% RSLogix 500 project PRJ_OUM_BAK033.RSS, saved by version 8.30.00.16 %
PROJECT "PRJ_OUM"    % processor: MicroLogix 1000 %

PROGRAM FILES
  LAD 2 "MAIN_PROG"  14 rungs
  LAD 3 "USER_FAULT"  1 rungs
  LAD 4 "HSC_INT"  1 rungs
  LAD 5 "STI_INT"  1 rungs
  LAD 6, 7, 8, 9, 10, 11, 12, 13, 14, 15, 16: only END

DATA FILES
  O0 OUTPUT  1 elements
  I1 INPUT  2 elements
  S2 STATUS  33 elements
  B3 BINARY  32 elements
  T4 TIMER  40 elements
  C5 COUNTER  32 elements
  R6 CONTROL  16 elements
  N7 INTEGER  105 elements

LADDER 2 "MAIN_PROG"
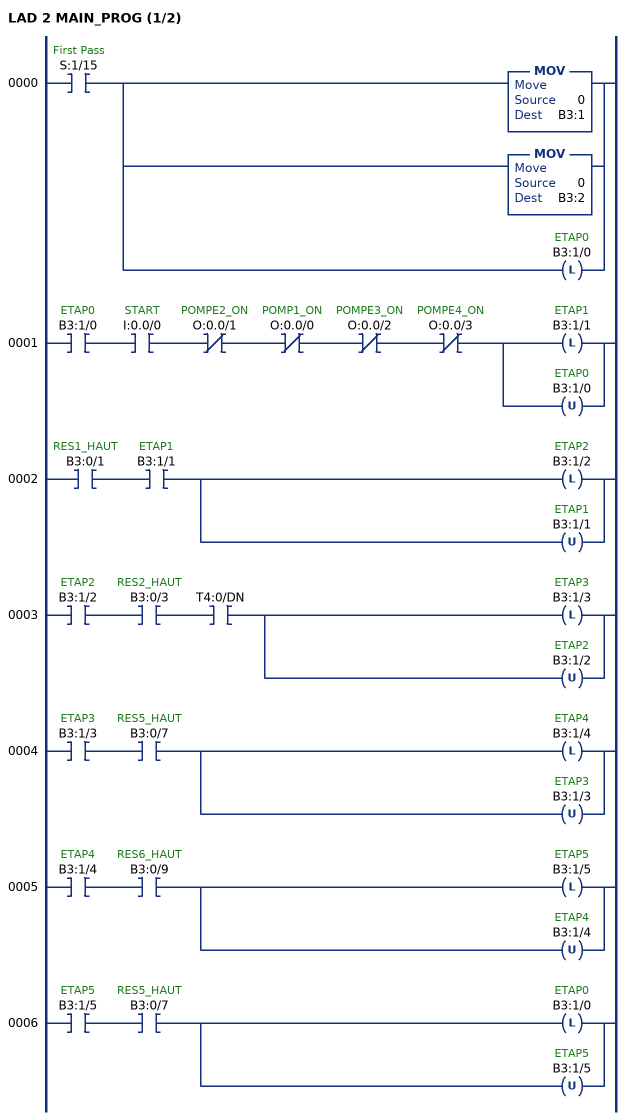
% Rung: 0 %
SOR XIC S:1/15 BST MOV 0 B3:1 NXB BST MOV 0 B3:2 NXB OTL B3:1/0 BND BND EOR
%   S:1/15  "First Pass" %
%   B3:1/0  ETAP0 %
% Rung: 1 %
SOR XIC B3:1/0 XIC I:0.0/0 XIO O:0.0/1 XIO O:0.0/0 XIO O:0.0/2 XIO O:0.0/3 BST OTL B3:1/1 NXB OTU B3:1/0 BND EOR
%   B3:1/0  ETAP0 %
%   I:0.0/0  START %
%   O:0.0/1  POMPE2_ON %
%   O:0.0/0  POMP1_ON %
%   O:0.0/2  POMPE3_ON %
%   O:0.0/3  POMPE4_ON %
%   B3:1/1  ETAP1 %
% Rung: 2 %
SOR XIC B3:0/1 XIC B3:1/1 BST OTL B3:1/2 NXB OTU B3:1/1 BND EOR
%   B3:0/1  RES1_HAUT %
%   B3:1/1  ETAP1 %
%   B3:1/2  ETAP2 %
% Rung: 3 %
SOR XIC B3:1/2 XIC B3:0/3 XIC T4:0/DN BST OTL B3:1/3 NXB OTU B3:1/2 BND EOR
%   B3:1/2  ETAP2 %
%   B3:0/3  RES2_HAUT %
%   B3:1/3  ETAP3 %
% Rung: 4 %
SOR XIC B3:1/3 XIC B3:0/7 BST OTL B3:1/4 NXB OTU B3:1/3 BND EOR
%   B3:1/3  ETAP3 %
%   B3:0/7  RES5_HAUT %
%   B3:1/4  ETAP4 %
% Rung: 5 %
SOR XIC B3:1/4 XIC B3:0/9 BST OTL B3:1/5 NXB OTU B3:1/4 BND EOR
%   B3:1/4  ETAP4 %
%   B3:0/9  RES6_HAUT %
%   B3:1/5  ETAP5 %
% Rung: 6 %
SOR XIC B3:1/5 XIC B3:0/7 BST OTL B3:1/0 NXB OTU B3:1/5 BND EOR
%   B3:1/5  ETAP5 %
%   B3:0/7  RES5_HAUT %
%   B3:1/0  ETAP0 %

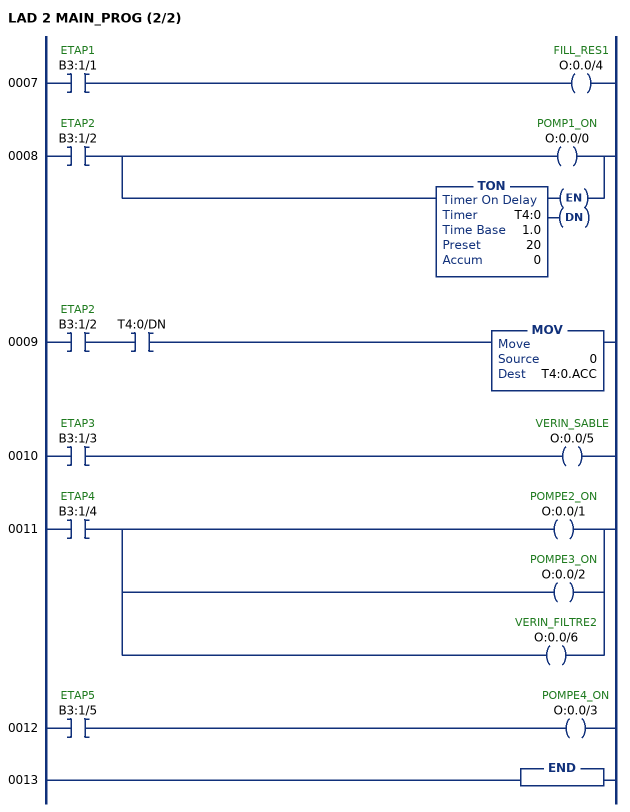
% Rung: 7 %
SOR XIC B3:1/1 OTE O:0.0/4 EOR
%   B3:1/1  ETAP1 %
%   O:0.0/4  FILL_RES1 %
% Rung: 8 %
SOR XIC B3:1/2 BST OTE O:0.0/0 NXB TON T4:0 1.0 20 0 BND EOR
%   B3:1/2  ETAP2 %
%   O:0.0/0  POMP1_ON %
% Rung: 9 %
SOR XIC B3:1/2 XIC T4:0/DN MOV 0 T4:0.ACC EOR
%   B3:1/2  ETAP2 %
% Rung: 10 %
SOR XIC B3:1/3 OTE O:0.0/5 EOR
%   B3:1/3  ETAP3 %
%   O:0.0/5  VERIN_SABLE %
% Rung: 11 %
SOR XIC B3:1/4 BST OTE O:0.0/1 NXB BST OTE O:0.0/2 NXB OTE O:0.0/6 BND BND EOR
%   B3:1/4  ETAP4 %
%   O:0.0/1  POMPE2_ON %
%   O:0.0/2  POMPE3_ON %
%   O:0.0/6  VERIN_FILTRE2 %
% Rung: 12 %
SOR XIC B3:1/5 OTE O:0.0/3 EOR
%   B3:1/5  ETAP5 %
%   O:0.0/3  POMPE4_ON %
% Rung: 13 %
SOR END EOR

OTHER DOCUMENTED ADDRESSES
  B3:0  B3
  B3:0/0  RES1_BAS
  B3:0/2  RES2_BAS
  B3:0/4  RES4_BAS
  B3:0/5  RES4_HAUT
  B3:0/6  RES5_BAS
  B3:0/8  RES6_BAS
  B3:0/10  RES7_BAS
  B3:0/11  RES7_HAUT
  B3:1/6  ETAP
  B3:1/7  ETAP6
  B3:1/8  ETAP8
  B3:1/9  ETAP9
  B3:1/10  ETAP10
  B3:1/11  ETAP11
  B3:1/12  ETAP12
  B3:1/13  ETAP13
  B3:1/14  ETAP14
  B3:1/15  ETAP15
  FF  
  POMP2_ON  

DATA TABLE (non-zero values as saved)
DATA B3
% B3:0 % 0X0055 0X0000 0X0000 0X0000 0X0000 0X0000 0X0000 0X0000 0X0000 0X0000
DATA T4
% .PRE .ACC %
% T4:0 % 20 0
